// TwinCAT 3 PLC project tc3base
// Title: Tc3_Base
// Company: Daniel Wiege
// ProjectVersion: 1.0.0.0
// ProgramVersion: 3.1.4026.21
// libraries:
//   Tc2_Standard, * (Beckhoff Automation GmbH)
//   Tc2_System, * (Beckhoff Automation GmbH)
// project tree:
//   1_Core/1_Object/ FB_Object.TcPOU (not stored), I_IgnoreInitRegistration.TcIO, I_Object.TcIO (not stored)
//   1_Core/2_Base/ FB_Base.TcPOU (not stored), I_Base.TcIO, I_FastCall.TcIO (not stored), I_MainCall.TcIO (not stored)
//   1_Core/3_Program/ FB_ProgramBase.TcPOU (not stored)
//   1_Core/4_DataContainer/ FB_DataContainer.TcPOU (not stored)
//   3_Management/ GVL_Manager.TcGVL
//   3_Management/InitManager/ FB_InitManager.TcPOU (not stored), I_InitManager.TcIO (not stored)
//   3_Management/ManagerBase/ FB_ManagerBase.TcPOU (not stored), FB_ManagerAdapter.TcPOU (not stored), FB_ManagerCollection.TcPOU (not stored), I_Manager.TcIO (not stored)
//   3_Management/LogManager/ FB_LogManager.TcPOU (not stored), FB_Logger.TcPOU (not stored)
//   Par/ Par_Core.TcGVL, Par_InitManager.TcGVL, Par_Manager.TcGVL
//   Project Information/ F_GetCompany.TcPOU, F_GetTitle.TcPOU, F_GetVersion.TcPOU
//   Version/ Global_Version.TcGVL

// ---- 3_Management/GVL_Manager.TcGVL
{attribute 'qualified_only'}
{attribute 'global_init_slot' := '40500'}
VAR_GLOBAL
	Collection				: FB_ManagerCollection(0);
	Managers				: FB_ManagerAdapter(0);
END_VAR

// ---- Par/Par_Core.TcGVL
{attribute 'qualified_only'}
VAR_GLOBAL CONSTANT
	MaxAmountProgramChildren				: UINT := 10;
END_VAR

// ---- Par/Par_InitManager.TcGVL
{attribute 'qualified_only'}
VAR_GLOBAL CONSTANT
	MaxAmountObject				: UINT := 10000;
END_VAR

// ---- Par/Par_Manager.TcGVL
{attribute 'qualified_only'}
VAR_GLOBAL CONSTANT
	MaxAmountManagers				: UINT := 10;
END_VAR

// ---- Version/Global_Version.TcGVL
{attribute 'TcGenerated'}
{attribute 'no-analysis'}
{attribute 'linkalways'}
// This function has been automatically generated from the project information.
VAR_GLOBAL CONSTANT
	{attribute 'const_non_replaced'}
	stLibVersion_Tc3_Base : ST_LibVersion := (iMajor := 1, iMinor := 0, iBuild := 0, iRevision := 0, nFlags := 0, sVersion := '1.0.0.0');
END_VAR

// ---- 1_Core/1_Object/I_IgnoreInitRegistration.TcIO
INTERFACE I_IgnoreInitRegistration EXTENDS __System.IQueryInterface

END_INTERFACE

// ---- 1_Core/2_Base/I_Base.TcIO
INTERFACE I_Base EXTENDS I_Object, I_FastCall, I_MainCall

END_INTERFACE

// ---- Project Information/F_GetCompany.TcPOU
// This function has been automatically generated from the project information.
{attribute 'signature_flag' := '1073741824'}
{attribute 'TcGenerated'}
{attribute 'no-analysis'}
FUNCTION F_GetCompany : WSTRING
VAR_INPUT
	
END_VAR

F_GetCompany := "Daniel Wiege";

END_FUNCTION

// ---- Project Information/F_GetTitle.TcPOU
// This function has been automatically generated from the project information.
{attribute 'signature_flag' := '1073741824'}
{attribute 'TcGenerated'}
{attribute 'no-analysis'}
FUNCTION F_GetTitle : WSTRING
VAR_INPUT
	
END_VAR

F_GetTitle := "Tc3_Base";

END_FUNCTION

// ---- Project Information/F_GetVersion.TcPOU
// This function has been automatically generated from the project information.
{attribute 'signature_flag' := '1073741824'}
{attribute 'TcGenerated'}
{attribute 'no-analysis'}
FUNCTION F_GetVersion : ST_LibVersion
VAR_INPUT
	
END_VAR

F_GetVersion.iMajor := 1;
F_GetVersion.iMinor := 0;
F_GetVersion.iBuild := 0;
F_GetVersion.iRevision := 0;
F_GetVersion.sVersion := '1.0.0.0';
F_GetVersion.nFlags := 0;

END_FUNCTION
